Staubli VAL3: helpers.pjx

--- helpers.pjx ---
Parameters version=s8.13.1Cs9_BS2800 stackSize=5000 millimeterUnit=true
Program file=allBool.pgx
Program file=anyBool.pgx
Program file=bin2dec.pgx
Program file=bindRow.pgx
Program file=bool2num.pgx
Program file=colSum.pgx
Program file=compare.pgx
Program file=compareStr.pgx
Program file=countBool.pgx
Program file=countBool2D.pgx
Program file=countBool3D.pgx
Program file=extractCol.pgx
Program file=extractGrid.pgx
Program file=extractNum.pgx
Program file=extractRow.pgx
Program file=extractRows.pgx
Program file=max_.pgx
Program file=mergeList.pgx
Program file=mergeVectors.pgx
Program file=min_.pgx
Program file=num2bool.pgx
Program file=printBool.pgx
Program file=printNum.pgx
Program file=printNum2d.pgx
Program file=printStr.pgx
Program file=range.pgx
Program file=readFile.pgx
Program file=repeat.pgx
Program file=rowSum.pgx
Program file=start.pgx
Program file=stop.pgx
Program file=uniqueNum.pgx
Program file=uniqueStr.pgx
Program file=vec2num.pgx
Program file=vecMax.pgx
Data file=helpers.dtx

--- helpers.dtx ---
public string sLetters[26]
  [0] = "a"
  [1] = "b"
  [2] = "c"
  [3] = "d"
  [4] = "e"
  [5] = "f"
  [6] = "g"
  [7] = "h"
  [8] = "i"
  [9] = "j"
  [10] = "k"
  [11] = "l"
  [12] = "m"
  [13] = "n"
  [14] = "o"
  [15] = "p"
  [16] = "q"
  [17] = "r"
  [18] = "s"
  [19] = "t"
  [20] = "u"
  [21] = "v"
  [22] = "w"
  [23] = "x"
  [24] = "y"
  [25] = "z"
public string sLETTERS[26]
  [0] = "A"
  [1] = "B"
  [2] = "C"
  [3] = "D"
  [4] = "E"
  [5] = "F"
  [6] = "G"
  [7] = "H"
  [8] = "I"
  [9] = "J"
  [10] = "K"
  [11] = "L"
  [12] = "M"
  [13] = "N"
  [14] = "O"
  [15] = "P"
  [16] = "Q"
  [17] = "R"
  [18] = "S"
  [19] = "T"
  [20] = "U"
  [21] = "V"
  [22] = "W"
  [23] = "X"
  [24] = "Y"
  [25] = "Z"
num nTest[5]
bool bResult
bool bError
bool bResult2
num nResult
string sStringBuffer
num nTest2[5]
num nMatrix[3 4]
num nResult2D[1 1]
num nResult_2[1 1]
num nRowResult
string sResult

--- start.pgx ---
program start()
  local num l_nBin[3]
  local num l_nRes
  local num l_nRows
  local num l_nCols
  local num l_nCounter
  local num l_nIndices[2]
  local string l_sString[10]
begin

  ? "## test num2Bool"
  ? "nTest[0] = nTest[1] = nTest[4] = 1"
  nTest[0] = nTest[1] = nTest[4] = 1

  call num2bool(nTest, bResult, bError)
  call printBool(bResult)

  ? "## test countBool"
  call countBool(bResult,nResult)
  call printNum(nResult)

  ? "## test allBool"
  call allBool(bResult, bResult2)
  call printBool(bResult2)

  ? "## test allBool"
  ? "nTest[2] = nTest[3] = 1"
  nTest[2] = nTest[3] = 1
  call num2bool(nTest, bResult, bError)
  call allBool(bResult, bResult2)
  call printBool(bResult2)

  ? "## test countBool"
  call countBool(bResult,nResult)
  call printNum(nResult)

  ? "## test anyBool TRUE"
  call anyBool(bResult, "TRUE",bResult2)
  call printBool(bResult2)

  ? "## test anyBool FALSE"
  call anyBool(bResult, "FALSE",bResult2)
  call printBool(bResult2)

  ? "## test bool2num"
  call bool2num(bResult, nResult, bError)
  call printNum(nResult)

  ? "## test bool2num"
  ? "nTest[0] = nTest[1] = nTest[4] = 0"
  nTest[0] = nTest[1] = nTest[4] = 0
  call num2bool(nTest, bResult, bError)
  call bool2num(bResult, nResult, bError)
  call printNum(nResult)

  ? "## test bin2dec"
  ? "nTest"
  l_nBin[0] = 1
  l_nBin[1] = 0
  l_nBin[2] = 0

  call bin2dec(l_nBin, l_nRes)
  call printNum(l_nRes)

  ? "## test mergeVectors"
  nTest2[0] = 5
  nTest2[1] = -3
  nTest2[2] = 10
  nTest2[4] = -1

  call mergeVectors(nTest, nTest2, nResult)
  call printNum(nResult)

  ? "## test colSum"
  for l_nRows = 0 to size(nMatrix,1)-1
    for l_nCols = 0 to size(nMatrix,2)-1
      nMatrix[l_nRows,l_nCols] = l_nCounter
      l_nCounter = l_nCounter +1
    endFor
  endFor

  // 0 1  2  3
  // 4 5  6  7
  // 8 9 10 11

  ? "## Matrix to analyse:"
  call printNum2d(nMatrix)

  call colSum(nMatrix, nResult)
  call printNum(nResult)

  ? "## test rowSum"
  call rowSum(nMatrix, nResult)
  call printNum(nResult)

  ? "## test extractRow"
  call extractRow(nMatrix, 2, nResult)
  call printNum(nResult)

  ? "## test extractRows"
  l_nIndices[0] = 2
  l_nIndices[1] = 1
  call extractRows(nMatrix, l_nIndices, nResult2D)
  call printNum2d(nResult2D)

  ? "## test extractCol"
  call extractCol(nMatrix, 3, nResult)
  call printNum(nResult)

  ? "## test extractGrid: rows"
  call extractGrid(nMatrix, 1, 2,0,nResult2D)
  call printNum2d(nResult2D)

  ? "## test extractGrid: cols"
  call extractGrid(nMatrix, 2, 3,0,nResult2D)
  call printNum2d(nResult2D)

  ? "## test repeat(nTest2,3)"
  call repeat(nTest2,3, nResult)
  call printNum(nResult)

  ? "## test uniqueStr()"
  l_sString[0] = "A"
  l_sString[1] = "B"
  l_sString[2] = "C"
  l_sString[3] = "A"
  l_sString[4] = "B"
  l_sString[5] = "B"
  l_sString[6] = "a"
  l_sString[7] = "D"
  l_sString[8] = "V"
  l_sString[9] = "G"

  call uniqueStr(l_sString, sResult)
  call printStr(sResult)


end

--- allBool.pgx ---
public program allBool(bool& x_bInput[], bool& x_bResult)
  local num l_nLength
  local num l_nElement
begin

  l_nLength = size(x_bInput)
  x_bResult = false

  for l_nElement = 0 to l_nLength-1
    if x_bInput[l_nElement] == false
      x_bResult = false
      return
    else
      x_bResult = true
    endIf
  endFor

end

--- anyBool.pgx ---
public program anyBool(bool& x_bInput[], string x_sBool, bool& x_bResult)
  local num l_nLength
  local num l_nElement
begin

  l_nLength = size(x_bInput)
  x_bResult = false

  for l_nElement = 0 to l_nLength-1
    if x_bInput[l_nElement] == false
      if x_sBool == "false" or x_sBool == "False" or x_sBool == "FALSE"
        x_bResult = true
        return
      elseIf x_sBool == "true" or x_sBool == "True" or x_sBool == "TRUE"
        x_bResult = false
      endIf
    elseIf x_bInput[l_nElement] == true
      if x_sBool == "false" or x_sBool == "False" or x_sBool == "FALSE"
        x_bResult = false
      elseIf x_sBool == "true" or x_sBool == "True" or x_sBool == "TRUE"
        x_bResult = true
        return
      endIf
    endIf
  endFor


end

--- bin2dec.pgx ---
public program bin2dec(num& x_nInput[], num& x_nResult)
  local num l_nElement
begin
  x_nResult = 0

  for l_nElement = 0 to size(x_nInput)-1
    x_nResult = x_nResult + x_nInput[l_nElement]*power(2,size(x_nInput) -1-l_nElement)
  endFor

end

--- bindRow.pgx ---
public program bindRow()
begin
end

--- bool2num.pgx ---
public program bool2num(bool& x_bInput[], num& x_nResult[], bool& x_bError)
  local num l_nLength
  local num l_nElement
begin

  x_bError = false
  l_nLength = size(x_bInput)
  x_nResult = 0
  resize(x_nResult, 1, l_nLength)

  for l_nElement = 0 to l_nLength-1
    if x_bInput[l_nElement] == true
      x_nResult[l_nElement] = 1
    elseIf x_bInput[l_nElement] == false
      x_nResult[l_nElement] = 0
    else
      x_bError = true
    endIf
  endFor

end

--- colSum.pgx ---
public program colSum(num& x_nInput[] (dimensions=2), num& x_nResult[])
  local num l_nCols
  local num l_nRows
  local num l_nElement[2]
begin

  l_nRows = size(x_nInput,1)
  l_nCols = size(x_nInput,2)

  resize(x_nResult,1,1)
  x_nResult = 0
  resize(x_nResult,1,l_nCols)

  for l_nElement[0] = 0 to l_nCols-1
    for l_nElement[1] = 0 to l_nRows-1
      x_nResult[l_nElement[0]] = x_nResult[l_nElement[0]] + x_nInput[l_nElement[1],l_nElement[0]]
    endFor
  endFor



end

--- compare.pgx ---
public program compare(num& x_nInput[], string x_sSign, num x_nCompareTo, bool& x_bResult[])
  local num l_nLength
  local num l_nElement
begin

  l_nLength = size(x_nInput)
  x_bResult[0] = false
  resize(x_bResult,1,l_nLength)

  switch x_sSign
    case ">"
      for l_nElement = 0 to l_nLength-1
        if x_nInput[l_nElement] > x_nCompareTo
          x_bResult[l_nElement] = true
        else
          x_bResult[l_nElement] = false
        endIf
      endFor
    break
    case ">="
      for l_nElement = 0 to l_nLength-1
        if x_nInput[l_nElement] >= x_nCompareTo
          x_bResult[l_nElement] = true
        else
          x_bResult[l_nElement] = false
        endIf
      endFor
    break
    case "<"
      for l_nElement = 0 to l_nLength-1
        if x_nInput[l_nElement] < x_nCompareTo
          x_bResult[l_nElement] = true
        else
          x_bResult[l_nElement] = false
        endIf
      endFor
    break
    case "<="
      for l_nElement = 0 to l_nLength-1
        if x_nInput[l_nElement] <= x_nCompareTo
          x_bResult[l_nElement] = true
        else
          x_bResult[l_nElement] = false
        endIf
      endFor
    break
    case "=="
      for l_nElement = 0 to l_nLength-1
        if x_nInput[l_nElement] == x_nCompareTo
          x_bResult[l_nElement] = true
        else
          x_bResult[l_nElement] = false
        endIf
      endFor
    break
  endSwitch
end

--- compareStr.pgx ---
public program compareStr(string& x_sInput[], string x_sCompareTo, bool& x_bResult[])
  local num l_nLength
  local num l_nElement
begin

  l_nLength = size(x_sInput)
  x_bResult[0] = false
  resize(x_bResult,1,l_nLength)

  for l_nElement = 0 to l_nLength-1
    if x_sInput[l_nElement] == x_sCompareTo
      x_bResult[l_nElement] = true
    else
      x_bResult[l_nElement] = false
    endIf
  endFor
end

--- countBool.pgx ---
public program countBool(bool& x_bInput[], num& x_nResult)
  local num l_nLength
  local num l_nElement
begin

  l_nLength = size(x_bInput)
  x_nResult = 0

  for l_nElement = 0 to l_nLength-1
    if x_bInput[l_nElement] == true
      x_nResult = x_nResult+1
    endIf
  endFor

end

--- countBool2D.pgx ---
public program countBool2D(bool& x_bInput[] (dimensions=2), num& x_nResult)
  local num l_nElement
  local num l_nDim[2]
begin

  x_nResult = 0

  for l_nDim[0] = 0 to size(x_bInput,1)-1
    for l_nDim[1] = 0 to size(x_bInput,2)-1
        if x_bInput[l_nDim[0], l_nDim[1]] == true
          x_nResult = x_nResult+1
        endIf
    endFor
  endFor

end

--- countBool3D.pgx ---
public program countBool3D(bool& x_bInput[] (dimensions=3), num& x_nResult)
  local num l_nElement
  local num l_nDim[3]
begin

  x_nResult = 0

  for l_nDim[0] = 0 to size(x_bInput,1)-1
    for l_nDim[1] = 0 to size(x_bInput,2)-1
      for l_nDim[2] = 0 to size(x_bInput,3)-1
        if x_bInput[l_nDim[0], l_nDim[1], l_nDim[2]] == true
          x_nResult = x_nResult+1
        endIf
      endFor
    endFor
  endFor

end

--- extractCol.pgx ---
public program extractCol(num& x_nInput[] (dimensions=2), num x_nCol, num& x_nResult[])
  local num l_nCol
  local num l_nCounter
  local num l_nRow
begin

  resize(x_nResult,1,1)
  x_nResult = 0
  resize(x_nResult,1, size(x_nInput,1))

  l_nCounter = 0
  for l_nRow = 0 to size(x_nInput,1)-1
    x_nResult[l_nCounter] = x_nInput[l_nRow,x_nCol]
    l_nCounter = l_nCounter +1
  endFor

end

--- extractGrid.pgx ---
public program extractGrid(num& x_nInput[] (dimensions=2), num x_nDimension, num x_nFrom, num x_nTo, num& x_nResult[] (dimensions=2))
  local num l_nX
  local num l_nY
  local num l_nCounter
  local num l_nStep
begin

  resize(x_nResult,1,1)
  resize(x_nResult,2,1)
  x_nResult[0,0] = -999999


  l_nCounter = 0
  if x_nDimension == 1
    resize(x_nResult,1,abs(x_nTo-x_nFrom)+1)
    resize(x_nResult,2,size(x_nInput,2))

    l_nStep = sel(x_nTo >= x_nFrom, 1, -1)

    for l_nX = x_nFrom to x_nTo step l_nStep
      for l_nY = 0 to size(x_nInput,2)-1
        x_nResult[l_nCounter, l_nY] = x_nInput[l_nX,l_nY]
      endFor
      l_nCounter = l_nCounter + 1
    endFor


  elseIf x_nDimension == 2

    resize(x_nResult,1, size(x_nInput,1))
    resize(x_nResult,2, abs(x_nTo-x_nFrom)+1)

    l_nStep = sel(x_nTo >= x_nFrom, 1, -1)

    for l_nY = x_nFrom to x_nTo step l_nStep
      for l_nX = 0 to size(x_nInput,1)-1
        x_nResult[l_nX, l_nCounter] = x_nInput[l_nX,l_nY]
      endFor
      l_nCounter = l_nCounter + 1
    endFor
  endIf

end

--- extractNum.pgx ---
public program extractNum(num& x_nInput[], num& x_nIndices[], num& x_nResult[])
  local num l_nElement
begin

  resize(x_nResult,1,size(x_nIndices))

  for l_nElement = 0 to size(x_nIndices)-1
    x_nResult[l_nElement] = x_nInput[x_nIndices[l_nElement]]
  endFor

end

--- extractRow.pgx ---
public program extractRow(num& x_nInput[] (dimensions=2), num x_nRow, num& x_nResult[])
  local num l_nCol
  local num l_nCounter
  local num l_nRow
begin

  resize(x_nResult,1,1)
  x_nResult = 0
  resize(x_nResult,1, size(x_nInput,2))

  l_nCounter=0
  for l_nCol = 0 to size(x_nInput,2)-1
    x_nResult[l_nCounter] = x_nInput[x_nRow,l_nCol]
    l_nCounter = l_nCounter +1
  endFor

end

--- extractRows.pgx ---
public program extractRows(num& x_nInput[] (dimensions=2), num& x_nIndices[], num& x_nResult[] (dimensions=2))
  local num l_nCol
  local num l_nCounter
  local num l_nRow
begin

  resize(x_nResult,1,1)
  resize(x_nResult,2,1)
  x_nResult[0,0] = 0
  resize(x_nResult,1, size(x_nIndices))
  resize(x_nResult,2, size(x_nInput,2))

  for l_nRow = 0 to size(x_nIndices)-1
    for l_nCol = 0 to size(x_nInput,2)-1
      x_nResult[l_nRow, l_nCol] = x_nInput[x_nIndices[l_nRow],l_nCol]
    endFor
  endFor

end

--- max_.pgx ---
public program max_(num& x_nInput[], num& x_nResult)
  local num l_nElement
begin

  x_nResult = -99999
  for l_nElement = 0 to size(x_nInput)-1
    x_nResult = max(x_nResult, x_nInput[l_nElement])
  endFor

end

--- mergeList.pgx ---
public program mergeList()
begin
end

--- mergeVectors.pgx ---
public program mergeVectors(num& x_nInput_1[], num& x_nInput_2[], num& x_nResult[])
  local num l_nLength[2]
  local num l_nElement
begin

  l_nLength[0] = size(x_nInput_1)
  l_nLength[1] = size(x_nInput_2)
  resize(x_nResult,1,1)
  x_nResult[0] = 0
  resize(x_nResult,1,l_nLength[0]+l_nLength[1])

  // combine the two inputs
  for l_nElement = 0 to size(x_nResult)-1
    if l_nElement < l_nLength[0]
      x_nResult[l_nElement] = x_nInput_1[l_nElement]
    else
      x_nResult[l_nElement] = x_nInput_2[l_nElement-l_nLength[0]]
    endIf

  endFor

end

--- min_.pgx ---
public program min_(num& x_nInput[], num& x_nResult)
  local num l_nElement
begin

  x_nResult = 99999
  for l_nElement = 0 to size(x_nInput)-1
    x_nResult = min(x_nResult, x_nInput[l_nElement])
  endFor

end

--- num2bool.pgx ---
public program num2bool(num& x_nInput[], bool& x_bResult[], bool& x_bError)
  local num l_nLength
  local num l_nElement
begin

  x_bError = false
  l_nLength = size(x_nInput)
  x_bResult = false
  resize(x_bResult, 1,l_nLength)

  for l_nElement = 0 to l_nLength-1
    if x_nInput[l_nElement] == 0
      x_bResult[l_nElement] = false
    elseIf x_nInput[l_nElement] == 1
      x_bResult[l_nElement] = true
    else
      x_bError = true
    endIf
  endFor

end

--- printBool.pgx ---
public program printBool(bool& x_bInput[])
  local num l_nElement
  local num l_nLength
begin

  l_nLength = size(x_bInput)

  for l_nElement = 0 to l_nLength-1
    ? x_bInput[l_nElement]
  endFor

end

--- printNum.pgx ---
public program printNum(num& x_nInput[])
  local num l_nElement
  local num l_nLength
begin

  l_nLength = size(x_nInput)

  for l_nElement = 0 to l_nLength-1
    ? x_nInput[l_nElement]
  endFor

end

--- printNum2d.pgx ---
public program printNum2d(num& x_nInput[] (dimensions=2))
  local num l_nElement
  local num l_nLength
  local num l_nRow
  local num l_RowResult
  local string l_sRow
begin

  for l_nRow = 0 to size(x_nInput,1)-1
    call extractRow(x_nInput, l_nRow, nRowResult)
    l_sRow = ""
    for l_nElement = 0 to size(nRowResult)-1
      l_sRow = l_sRow + toString(".3", nRowResult[l_nElement])
    endFor
    ? l_sRow
    endFor

end

--- printStr.pgx ---
public program printStr(string& x_sInput[])
  local num l_nElement
  local num l_nLength
begin

  l_nLength = size(x_sInput)

  for l_nElement = 0 to l_nLength-1
    ? x_sInput[l_nElement]
  endFor

end

--- range.pgx ---
public program range(num x_nStart, num x_nEnd, num x_nStep, num& x_nResult[])
  local num l_nCoutner
  local num l_nElement
begin

  l_nCoutner = 0
  resize(x_nResult,1,1)
  x_nResult = 0

  for l_nElement = x_nStart to x_nEnd-1 step x_nStep
    l_nCoutner = l_nCoutner+1
    append(x_nResult)
    x_nResult[l_nCoutner] = l_nElement
  endFor

  delete(x_nResult[0])

end

--- readFile.pgx ---
public program readFile(string x_sFilename, string& x_sLine[])
  local num l_nFileHandler
  local num l_nReadLines
  local num l_nDataSize
  local string l_sLine
begin

  // Open file to write
  l_nFileHandler = $fileOpen(x_sFilename, "r")
  // init Buffer sLine
  resize(x_sLine, 1, 1)
  x_sLine = ""
  l_nDataSize = 0
  // read line by line
  do
    l_nReadLines = $fileGet(l_nFileHandler,l_sLine,1)
    if l_nReadLines > 0
      append(x_sLine)
      x_sLine[l_nDataSize] = l_sLine
    endIf
    l_nDataSize = l_nDataSize + 1
  until l_nReadLines == 0

  // remove last entry in x_sLine, because of "append" command before
  resize(x_sLine, 1, size(x_sLine)-1)
  // close file
  $fileClose(l_nFileHandler)

end

--- repeat.pgx ---
public program repeat(num& x_nInput[], num x_nTimes, num& x_nResult[])
  local num l_nElement
  local num l_nTimes
  local num l_nCounter
  local num l_nAppend
begin

  //rep(c(1,2,3),4) -> 1,2,3,1,2,3,1,2,3,1, 2, 3
  //                   0,1,2,3,4,5,6,7,8,9,10,11

  resize(x_nResult,1,size(x_nInput)*x_nTimes)

  for l_nElement = 1 to x_nTimes
    for l_nAppend = 0 to size(x_nInput)-1
      x_nResult[l_nCounter+l_nAppend] = x_nInput[l_nAppend]
    endFor
    l_nCounter = l_nCounter+size(x_nInput)
  endFor


end

--- rowSum.pgx ---
public program rowSum(num& x_nInput[] (dimensions=2), num& x_nResult[])
  local num l_nCols
  local num l_nRows
  local num l_nElement[2]
begin

  l_nRows = size(x_nInput,1)
  l_nCols = size(x_nInput,2)

  resize(x_nResult,1,1)
  x_nResult = 0
  resize(x_nResult,1,l_nRows)

  for l_nElement[0] = 0 to l_nRows-1
    for l_nElement[1] = 0 to l_nCols-1
      x_nResult[l_nElement[0]] = x_nResult[l_nElement[0]] + x_nInput[l_nElement[0],l_nElement[1]]
    endFor
  endFor



end

--- uniqueNum.pgx ---
public program uniqueNum(num& x_nInput[], num& x_nResult[])
  local num l_nCoutner
  local num l_nElement
  local num l_nLength
  local string l_sString
  local num l_nBuffer
begin

//  l_nLength = size(x_sInput)
//  l_nCoutner = 0
//  resize(x_sResult,1,1)
//  resize(sStringBuffer,1,1)

//  for l_nElement = 0 to l_nLength-1

//    if l_nElement = 0
//      append(x_sResult)
//      x_sResult[size(x_sResult)-1] = x_nInput[l_nElement]
//    else

//      for l_nBuffer = 0 to size(x_sResult)-1
//        if x_sInput[l_nElement] != x_sResult[l_nBuffer]
//          append(x_sResult)
//          x_sResult[size(x_sResult)-1] = x_nInput[l_nElement]
//        endIf

//      endFor

//    endIf

//  endFor

//  delete(x_sResult[0])

end

--- uniqueStr.pgx ---
public program uniqueStr(string& x_sInput[], string& x_sResult[])
  local num l_nCoutner
  local num l_nElement
  local num l_nLength
  local string l_sString
  local num l_nBuffer
  local bool l_bDone
  local bool l_bFound
  local num l_nMarker
begin

  l_nLength = size(x_sInput)
  l_nCoutner = 0
  resize(x_sResult,1,1)

  for l_nElement = 0 to l_nLength-1
    l_bFound = false
    if l_nElement == 0
      append(x_sResult)
      x_sResult[size(x_sResult)-1] = x_sInput[l_nElement]
    else

      for l_nBuffer = 0 to size(x_sResult)-1
        if x_sInput[l_nElement] != x_sResult[l_nBuffer]
          l_bFound = false
        else
          // break out of for-loop
          l_bFound = true
          l_nBuffer = size(x_sResult)+1
          l_nMarker = l_nBuffer
        endIf

      endFor

      if l_bFound == false
        append(x_sResult)
        x_sResult[size(x_sResult)-1] = x_sInput[l_nElement]
      endIf

   endIf

  endFor

  delete(x_sResult[0])

end

--- vec2num.pgx ---
public program vec2num(string& x_sInput[], num& x_nResult[])
  local num l_nLength
  local num l_nElement
  local string l_sCopy
  local num l_nValue
  local bool l_bSucces
  local num l_nSucessCounter
begin

  l_nLength = size(x_sInput)
  x_nResult[0] = 0
  resize(x_nResult,1,1)

  for l_nElement = 0 to l_nLength-1
    // copy element
    l_sCopy = x_sInput[l_nElement]
    toNum(l_sCopy, l_nValue, l_bSucces)
    if l_bSucces
      if l_nElement !=0
        append(x_nResult)
      endIf
      x_nResult[l_nSucessCounter] = l_nValue
      l_nSucessCounter = l_nSucessCounter +1
    endIf
  endFor

end

--- vecMax.pgx ---
public program vecMax(num& x_nInput[], num& x_nResult)
  local num l_nElement
  local num l_nMax
begin

  l_nMax = -999999
  for l_nElement = 0 to size(x_nInput)-1
    l_nMax = max(l_nMax, x_nInput[l_nElement])
  endFor

  x_nResult = l_nMax

end
